FUNCTION_BLOCK FB_WeightSorter
VAR_INPUT
	weight_input : REAL;
END_VAR
VAR_OUTPUT
	iPackageSize : INT;
	
	small : BOOL;
	medium : BOOL;
	large : BOOL;
END_VAR
VAR
END_VAR
VAR // added by the converter: edge detectors and wires of the graphical bodies
    _w1, _w2, _w3 : BOOL;
END_VAR

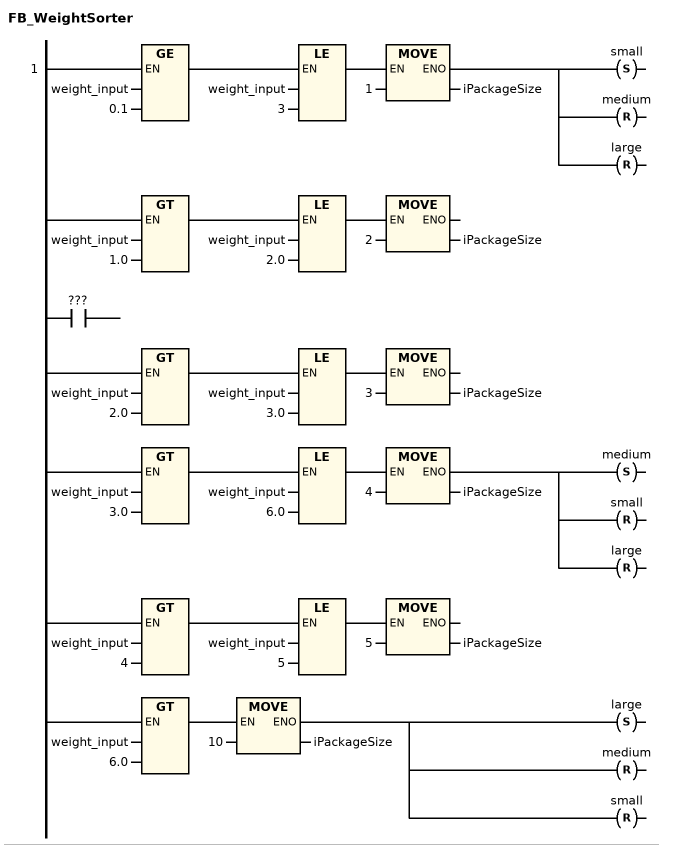
// NETWORK 1
_w1 := weight_input >= 0.1 AND weight_input <= 3;
IF _w1 THEN iPackageSize := 1; END_IF
small S= _w1;
medium R= _w1;
large R= _w1;
IF weight_input > 1.0 AND weight_input <= 2.0 THEN iPackageSize := 2; END_IF
IF weight_input > 2.0 AND weight_input <= 3.0 THEN iPackageSize := 3; END_IF
_w2 := weight_input > 3.0 AND weight_input <= 6.0;
IF _w2 THEN iPackageSize := 4; END_IF
medium S= _w2;
small R= _w2;
large R= _w2;
IF weight_input > 4 AND weight_input <= 5 THEN iPackageSize := 5; END_IF
_w3 := weight_input > 6.0;
IF _w3 THEN iPackageSize := 10; END_IF
large S= _w3;
medium R= _w3;
small R= _w3;

END_FUNCTION_BLOCK

(* stored: Version 1.1.0.1, ProductVersion 3.1.4024.13
   POU FB_WeightSorter: Id {9b7c85d3-252e-4f2a-8908-ccb4e0a8684d}, SpecialFunc None *)
